// TIA Portal V20 export
// export: Created 2026-04-11T06:02:29.8797724Z, ExportSetting WithDefaults, DisplayName Totally Integrated Automation Portal, DisplayVersion V20, DisplayName TIA Portal Openness, DisplayVersion V20, DisplayName TIA Portal Version Control Interface, DisplayVersion V20, DisplayName STEP 7 Professional, DisplayVersion V20, DisplayName STEP 7 Safety, DisplayVersion V20, DisplayName WinCC Basic/Comfort/Advanced, DisplayVersion V20, DisplayName WinCC Unified, DisplayVersion V20
TYPE "udtError_USSDrive"
// stored: IsFailsafeCompliant false
   STRUCT
      bLengthError { ExternalWritable := 'False'} : Bool;   // Length error in drive response
      bDataTypeError { ExternalWritable := 'False'} : Bool;   // Data type error
      bWordRequestError { ExternalWritable := 'False'} : Bool;   // Data type error - DWord or Real returned from Word request
      bDWordOrRealRequestError { ExternalWritable := 'False'} : Bool;   // Data type error - Word returned from DWord or Real request
      bChecksumError { ExternalWritable := 'False'} : Bool;   // Checksum error in drive response
      bAddressingError { ExternalWritable := 'False'} : Bool;   // Addressing error
      bSetpointError { ExternalWritable := 'False'} : Bool;   // Setpoint error
      bIncorrectDriveNumber { ExternalWritable := 'False'} : Bool;   // Incorrect drive number returned
      bInvalidLength { ExternalWritable := 'False'} : Bool;   // Invalid PZD length
      bInvalidBaudrate { ExternalWritable := 'False'} : Bool;   // The module does not support this transmission rate
      bRequestActive { ExternalWritable := 'False'} : Bool;   // A different request for this drive is currently active
      bNoResponse { ExternalWritable := 'False'} : Bool;   // The drive does not respond
      bParameterRequestError { ExternalWritable := 'False'} : Bool;   // The drive responds with an error message to a parameter request
      bParameterRequestAccessError { ExternalWritable := 'False'} : Bool;   // The drive responds with an access error message to a parameter request
      bNotInitialized { ExternalWritable := 'False'} : Bool;   // The drive was not initialized
      bNegativeAckRead { ExternalWritable := 'False'} : Bool;   // Negative acknowledgment when reading module
      bNegativeAckWrite { ExternalWritable := 'False'} : Bool;   // Negative acknowledgment when writing module
   END_STRUCT;
END_TYPE
